{attribute 'GeneratedUsingTerminal: EK1100-0000-0018'}
{attribute addProperty BoxType "EK1100-0000-0018"}
{attribute addProperty Id "Beckhoff_EKx9xxEK1122Beckhoff_EKx9xxEK1122_41BF98AA1154"}
{attribute addProperty CRC "917081774"}
{attribute addProperty Size "1154"}
TYPE Beckhoff_EKx9xx_36A98EAE EXTENDS EK1100_1FC0878B :
STRUCT
	{attribute addProperty Name "Beckhoff_EKx9xxEK1122"}
	Beckhoff_EKx9xxEK1122 : Beckhoff_EKx9xxEK1122_41BF98AA;
END_STRUCT
END_TYPE

(* stored: Version 1.2.0.0, ProductVersion 3.1.4024.9
   DUT Beckhoff_EKx9xx_36A98EAE: Id {a774f7e2-a899-4b8d-baaa-f006daf0c6a0} *)
